// TwinCAT 3 PLC project FIO
// ProgramVersion: 3.1.4023.0
// libraries:
//   Tc2_ModbusSrv, * (Beckhoff Automation GmbH)
//   Tc2_Standard, * (Beckhoff Automation GmbH)
//   Tc2_System, * (Beckhoff Automation GmbH)
//   Tc3_Module, * (Beckhoff Automation GmbH)
// project tree:
//   GVLs/ GVL.TcGVL
//   / PlcTask.TcTTO
//   POUs/ CONTROL.TcDUT, MAIN.TcPOU, ModbusReadInputs.TcPOU, ModbusWriteOutputs.TcPOU
// real-time tasks:
//   TASK PlcTask: cycle T#10ms, priority 20, ADS port 350

CONFIGURATION FIO
    RESOURCE PLC ON TwinCAT3
        TASK PlcTask(INTERVAL := T#10ms, PRIORITY := 20);
        PROGRAM MAIN WITH PlcTask : MAIN;
    END_RESOURCE
END_CONFIGURATION

// ---- POUs/CONTROL.TcDUT
{attribute 'qualified_only'}
{attribute 'strict'}
TYPE CONTROL :
(
	StartConveyor := 0000_0001,
	StopConveyor := 0000_0000
) BYTE;
END_TYPE

// ---- GVLs/GVL.TcGVL
{attribute 'qualified_only'}
VAR_GLOBAL
	
END_VAR

// ---- POUs/MAIN.TcPOU
PROGRAM MAIN
VAR
	fb_ReadInputs : ModbusReadInputs;
	fb_WriteOutputs : ModbusWriteOutputs;
	data: ARRAY [0..1] OF BYTE;
	bSensorEndConveyor: BOOL;
	bStartStopConveyor: ARRAY [0..1] OF BYTE := [2#0000_0001, 2#0000_0000];
END_VAR

fb_ReadInputs(Data=> data);
bSensorEndConveyor := data[0].0;

IF bSensorEndConveyor THEN
	fb_WriteOutputs(Data := CONTROL.StartConveyor);
//ELSIF NOT bSensorEndConveyor THEN
	//fb_WriteOutputs(Data := CONTROL.StopConveyor);	
END_IF;

END_PROGRAM

// ---- POUs/ModbusReadInputs.TcPOU
FUNCTION_BLOCK ModbusReadInputs

VAR_INPUT
	
END_VAR

VAR_OUTPUT
	Data : ARRAY [0..1] OF BYTE;
	bReadInputsBusy : BOOL;
    bReadInputsError : BOOL;
    nReadInputsErrorId : UDINT;
END_VAR

VAR
	fbReadInputs : FB_MBReadInputs;
END_VAR

fbReadInputs(
	sIPAddr := '127.0.0.1', // Is a string containing the IP address of the target device
	nTCPPort := 505, //Port number of the target device.
	nUnitID := 255, //  Identification number of a serial sub-network device. (Slave number)
	nQuantity := 16, // Number of digital inputs (data bits) to be read
	nMBAddr := 0, // Start address of the digital inputs to be read (bit offset).
	cbLength := SIZEOF(Data),
	pDestAddr := ADR(Data), // Contains the address of the destination buffer into which the data are to be read.
	bExecute := TRUE, // The function block is activated by a rising edge at this input.
	tTimeout := T#1S, // States the length of the timeout that may not be exceeded by execution of the ADS command.
	bBusy => bReadInputsBusy ,
	bError => bReadInputsError,
	nErrId => nReadInputsErrorId,
	cbRead => ,
);

// The FB_MBReadInputs get activated after a rising edge at bExecute input.
fbReadInputs(bExecute := FALSE);
fbReadInputs(bExecute := TRUE);

END_FUNCTION_BLOCK

// ---- POUs/ModbusWriteOutputs.TcPOU
FUNCTION_BLOCK ModbusWriteOutputs
VAR_INPUT
	Data : BYTE;
END_VAR
	
VAR_OUTPUT
	bBUSY : BOOL;
	bError : BOOL;
	nErrId : UDINT;
END_VAR

VAR
	fbwriteoutputs : FB_MBWriteCoils;
END_VAR

fbwriteoutputs(
	sIPAddr := '127.0.0.1', 
	nTCPPort := 505, 
	nUnitID := 255,
	nQuantity := 2,
	nMBAddr := 0, 
	cbLength := SIZEOF(Data),
	pSrcAddr := ADR(Data),
	bExecute := TRUE, 
	tTimeout := T#1S,
);

END_FUNCTION_BLOCK
